SUBAPPLICATION Uebung_004a2 (* mit E_MERGE *)
  (* Standard: 61499-2 *)
  (* Version 1.0, 2023-10-23, franz *)
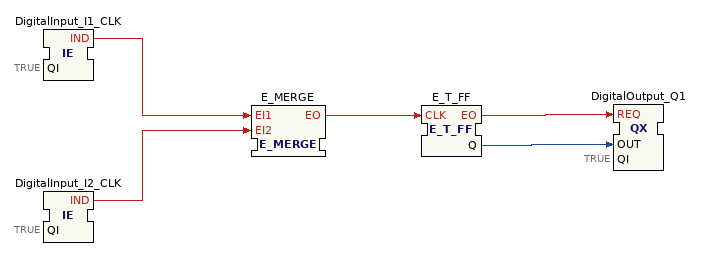
  FBS
    DigitalOutput_Q1 : QX(QI := TRUE);
    DigitalInput_I1_CLK : IE(QI := TRUE);
    E_T_FF : E_T_FF;
    E_MERGE : E_MERGE;
    DigitalInput_I2_CLK : IE(QI := TRUE);
  END_FBS
  EVENT_CONNECTIONS
    E_T_FF.EO TO DigitalOutput_Q1.REQ;
    DigitalInput_I1_CLK.IND TO E_MERGE.EI1;
    DigitalInput_I2_CLK.IND TO E_MERGE.EI2;
    E_MERGE.EO TO E_T_FF.CLK;
  END_CONNECTIONS
  DATA_CONNECTIONS
    E_T_FF.Q TO DigitalOutput_Q1.OUT;
  END_CONNECTIONS
END_SUBAPPLICATION
